FUNCTION_BLOCK CLNTRC_1 (* Wrapper for a CLIENT FB using the HTTP communciation protocol. Attempts to reconnect upon error. *)
  (* Standard: 61499-2 *)
  (* Version 0.0, 2017-09-05, 4DIAC-IDE, 4DIAC-Consortium *)
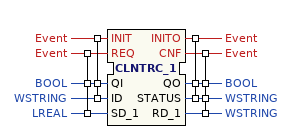
  EVENT_INPUT
    INIT WITH QI, ID; (* Initialization Request *)
    REQ WITH QI, SD_1; (* Normal Execution Request *)
  END_EVENT
  EVENT_OUTPUT
    INITO WITH QO, STATUS; (* Initialization Confirm *)
    CNF WITH QO, STATUS, RD_1; (* Execution Confirmation *)
  END_EVENT
  VAR_INPUT
    QI : BOOL; (* Input event qualifier *)
    ID : WSTRING; (* Connection Identifier *)
    SD_1 : LREAL; (* Input Data *)
  END_VAR
  VAR_OUTPUT
    QO : BOOL; (* Output event qualifier *)
    STATUS : WSTRING; (* Service Status *)
    RD_1 : WSTRING; (* Received Data *)
  END_VAR
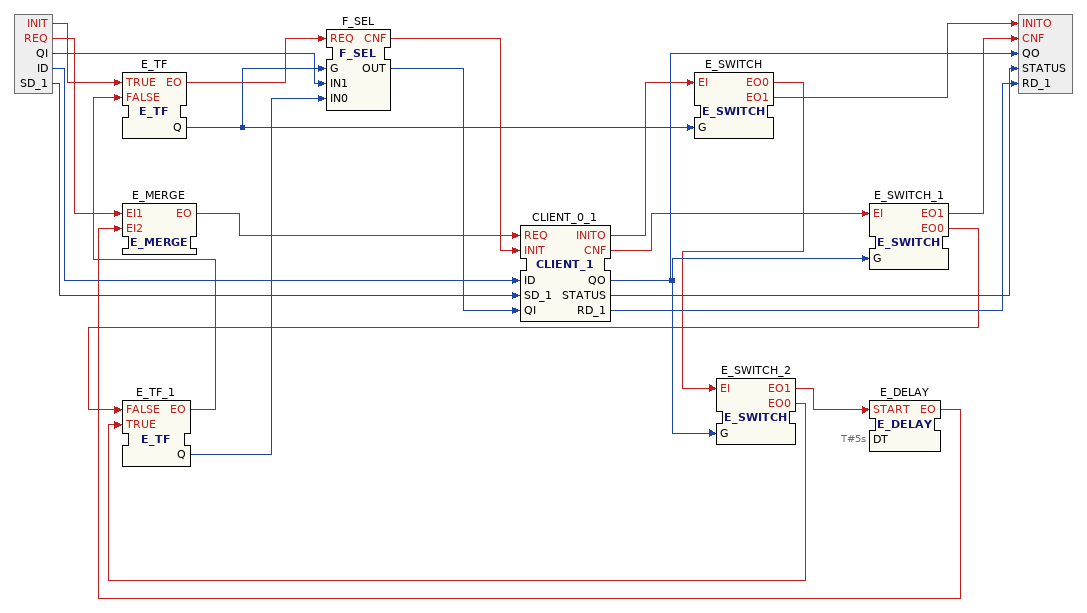
  FBS
    E_TF : E_TF;
    E_SWITCH : E_SWITCH;
    E_MERGE : E_MERGE;
    E_SWITCH_1 : E_SWITCH;
    E_SWITCH_2 : E_SWITCH;
    CLIENT_0_1 : CLIENT_1;
    E_DELAY : E_DELAY(DT := T#5s);
    E_TF_1 : E_TF;
    F_SEL : F_SEL;
  END_FBS
  EVENT_CONNECTIONS
    INIT TO E_TF.TRUE;
    REQ TO E_MERGE.EI1;
    E_SWITCH_1.EO1 TO CNF;
    E_SWITCH.EO0 TO E_SWITCH_2.EI;
    E_MERGE.EO TO CLIENT_0_1.REQ;
    CLIENT_0_1.INITO TO E_SWITCH.EI;
    CLIENT_0_1.CNF TO E_SWITCH_1.EI;
    E_DELAY.EO TO E_MERGE.EI2;
    E_SWITCH_2.EO1 TO E_DELAY.START;
    E_SWITCH_1.EO0 TO E_TF_1.FALSE;
    E_SWITCH.EO1 TO INITO;
    E_SWITCH_2.EO0 TO E_TF_1.TRUE;
    E_TF.EO TO F_SEL.REQ;
    F_SEL.CNF TO CLIENT_0_1.INIT;
    E_TF_1.EO TO E_TF.FALSE;
  END_CONNECTIONS
  DATA_CONNECTIONS
    E_TF.Q TO E_SWITCH.G;
    ID TO CLIENT_0_1.ID;
    CLIENT_0_1.QO TO E_SWITCH_1.G;
    CLIENT_0_1.QO TO E_SWITCH_2.G;
    CLIENT_0_1.QO TO QO;
    CLIENT_0_1.STATUS TO STATUS;
    CLIENT_0_1.RD_1 TO RD_1;
    SD_1 TO CLIENT_0_1.SD_1;
    E_TF.Q TO F_SEL.G;
    F_SEL.OUT TO CLIENT_0_1.QI;
    QI TO F_SEL.IN1;
    E_TF_1.Q TO F_SEL.IN0;
  END_CONNECTIONS
END_FUNCTION_BLOCK
